PROGRAM RunGrindingWheel
VAR
END_VAR

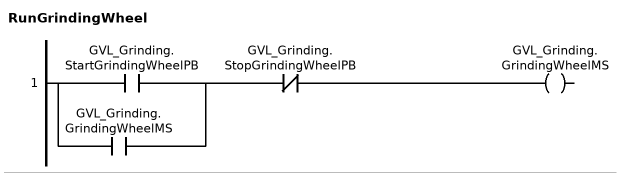
// NETWORK 1
GVL_Grinding.GrindingWheelMS := (GVL_Grinding.StartGrindingWheelPB OR GVL_Grinding.GrindingWheelMS) AND NOT GVL_Grinding.StopGrindingWheelPB;

END_PROGRAM

(* stored: Version 1.1.0.1, ProductVersion 3.1.4024.12
   POU RunGrindingWheel: Id {b63b43fa-8e36-408e-865a-bb277ea9fe78}, SpecialFunc None *)
